FUNCTION_BLOCK FB_S_Fuellstandsensor
VAR_INPUT
	I_iSignal			:INT;		// Messsignal des Sensors
	I_rHigh				:REAL;		// Oberer Schwellenwert für Prozess
	I_rLow				:REAL;		// Unterer Schwellenwert für Prozess
	I_rMax				:REAL;		// Skallierungswert -> Max-Wert 
	I_rMin				:REAL;		// Skallierungswert -> Min-Wert 
END_VAR

VAR_OUTPUT
	O_bStoerung			:BOOL;		// Befindet sich das Element in einem Error
	O_iStoerungID		:INT;		// Anzeigen von Störung über eine INT-Variable
END_VAR

VAR
	Messwert			:REAL;		// Wert für HMI
	GrenzeOben			:BOOL;		// Wert für HMI
	GrenzeUnten			:BOOL;		// Wert für HMI
END_VAR

Messwert := P_Messwert;
GrenzeOben := P_GrenzeOben;
GrenzeUnten := P_GrenzeUnten;

PROPERTY PUBLIC P_GrenzeOben : BOOL
GET
IF P_Messwert > I_rHigh THEN
	P_GrenzeOben := TRUE;
ELSE
	P_GrenzeOben := FALSE;
END_IF
END_GET
END_PROPERTY

PROPERTY PUBLIC P_GrenzeUnten : BOOL
GET
IF P_Messwert < I_rLow THEN
	P_GrenzeUnten := TRUE;
ELSE
	P_GrenzeUnten := FALSE;
END_IF
END_GET
END_PROPERTY

PROPERTY PUBLIC P_Messwert : REAL
GET
IF I_iSignal > 27648 OR I_iSignal < 0 THEN
	O_bStoerung := TRUE;
	O_iStoerungID := 04;
ELSE
	O_bStoerung := FALSE; 
END_IF

// Linearisierung des Wertes 
P_Messwert := INT_TO_REAL(I_iSignal) * (I_rMax-I_rMin) / 27648 + I_rMin;
END_GET
END_PROPERTY

END_FUNCTION_BLOCK

(* stored: Version 1.1.0.1, ProductVersion 3.1.4024.12
   POU FB_S_Fuellstandsensor: Id {67ce70cf-9cdd-4063-932f-0e6c679aeb25}, SpecialFunc None
   Property P_GrenzeOben: Id {f7a56a93-1bcc-4b2f-b2bf-9621efc6d809}
   Get Get: Id {b128aec4-3cc4-4a61-bcc9-2238cfb2a288}
   Property P_GrenzeUnten: Id {d7752ab2-f22c-45cb-8c81-2d3f67564794}
   Get Get: Id {e637b3d7-8ea9-4d2c-b6d9-a5d3192db478}
   Property P_Messwert: Id {6835c3d8-6b2c-4e92-aacc-80dd5e0395a0}
   Get Get: Id {f9bf7b4d-9263-4a2b-ad75-e3bdaeeaaccd} *)
